FUNCTION_BLOCK MovingAverageFilter
VAR_INPUT
	InputValue							:REAL;	
	tTaskCycleNumber					:INT;
	SampleNumber						:INT;
END_VAR
VAR_OUTPUT
	FilterValute						:REAL;
END_VAR
VAR
	i									:INT;	
	MainWorkingArra						:ARRAY[1..10] OF REAL;
	WorkingArraySum						:REAL;
	SumRange							:INT:=0;
	CycleNumber							:INT:=0;
END_VAR

FilterValute:=SEL(OnOrOffFilter(),InputValue,FilterValueMeth());

METHOD PRIVATE FilterValueMeth : real
IF SampleNumber=0 THEN
	SampleNumber:=1;
END_IF
CycleNumber:=CycleNumber+1;
IF CycleNumber>=tTaskCycleNumber THEN
	CycleNumber:=0;
	WorkingArraySum:=0;	
	SumRange:=SumRange+1;
	MainWorkingArra[SumRange]:=InputValue;
		FOR i:=1 TO SampleNumber BY 1 DO
			WorkingArraySum:=MainWorkingArra[i]+WorkingArraySum;
		END_FOR	
		IF SumRange=SampleNumber THEN
			SumRange:=0;
		END_IF		
END_IF
FilterValueMeth:=WorkingArraySum/SampleNumber;
END_METHOD

METHOD PRIVATE OnOrOffFilter : BOOL
VAR_INPUT
END_VAR
IF tTaskCycleNumber=0 OR tTaskCycleNumber=1 THEN
    OnOrOffFilter:=FALSE;
ELSE
    OnOrOffFilter:=TRUE;
END_IF
END_METHOD

END_FUNCTION_BLOCK

(* stored: Version 1.1.0.1, ProductVersion 3.1.4024.12
   POU MovingAverageFilter: Id {4977d736-bb6f-4b1e-953a-c5f4918e3ef7}, SpecialFunc None
   Method FilterValueMeth: Id {5ff84ea0-22d8-4944-8d69-e47a9dafbf8a}
   Method OnOrOffFilter: Id {9616f11e-b025-4a8e-ae2b-ccee7e4e1aea} *)
